// TwinCAT 3 PLC project PLC1
// ProgramVersion: 3.1.4026.23
// libraries:
//   Tc2_Standard, * (Beckhoff Automation GmbH)
//   Tc2_System, * (Beckhoff Automation GmbH)
// project tree:
//   / IsolatedCoreTask.TcTTO, SharedCoreTask.TcTTO
//   POUs/ F_CreateCPULoad.TcPOU, PRG_SharedCore.TcPOU, PRG_IsolatedCore.TcPOU
// real-time tasks:
//   TASK SharedCoreTask: cycle T#10ms, priority 1, ADS port 351
//   TASK IsolatedCoreTask: cycle T#10ms, priority 2, ADS port 352

CONFIGURATION PLC1
    RESOURCE PLC ON TwinCAT3
        TASK IsolatedCoreTask(INTERVAL := T#10ms, PRIORITY := 2);
        TASK SharedCoreTask(INTERVAL := T#10ms, PRIORITY := 1);
        PROGRAM PRG_IsolatedCore WITH IsolatedCoreTask : PRG_IsolatedCore;
        PROGRAM PRG_SharedCore WITH SharedCoreTask : PRG_SharedCore;
    END_RESOURCE
END_CONFIGURATION

// ---- POUs/PRG_IsolatedCore.TcPOU
PROGRAM PRG_IsolatedCore
VAR
END_VAR

F_CreateCPULoad();

END_PROGRAM

// ---- POUs/F_CreateCPULoad.TcPOU
FUNCTION F_CreateCPULoad
VAR_INPUT
	nIterations : DINT := 300000; (* Tune this to adjust load *)
END_VAR

VAR
	iIter  : DINT;
	fAccum : LREAL := 0.0;
END_VAR

FOR iIter := 1 TO nIterations DO
	fAccum := fAccum + SQRT(DINT_TO_LREAL(iIter));
END_FOR

END_FUNCTION

// ---- POUs/PRG_SharedCore.TcPOU
PROGRAM PRG_SharedCore
VAR
END_VAR

F_CreateCPULoad();

END_PROGRAM
